//==============================================================
// 12) Servo enable and magnetic brake control
//==============================================================
// EN: Zero the movement request immediately, command quick stop and keep the
//     servo enabled only for the configured shutdown delay.
//     Drive-ready feedback is not used to avoid a circular enable dependency.
// PT: Zera a solicitação de movimento imediatamente, comanda o quick stop e
//     mantém o servo habilitado apenas durante o atraso configurado de desligamento.
//     O retorno de drive pronto não é usado para evitar dependência circular.
elevatorDriveEnableRequest :=
    systemRunEnable AND
    safetyCircuitOk;

tofElevatorDriveDisableDelay(
    IN := elevatorDriveEnableRequest,
    PT := machineConfig.elevatorDriveDisableDelay
);

elevatorDriveEnable :=
    tofElevatorDriveDisableDelay.Q;

elevatorQuickStop :=
    NOT elevatorDriveEnableRequest AND
    tofElevatorDriveDisableDelay.Q;

elevatorMoveRequest :=
    systemRunEnable AND
    safetyCircuitOk AND
    elevatorDriveOk AND
    NOT elevatorFault AND
    (ABS(elevatorSignedSpeedRefMmps) > 0.0);

IF elevatorMoveRequest THEN

    elevatorBrakeReleaseRequest := TRUE;
    tonElevatorBrakeHoldDelay(IN := FALSE);

ELSE

    IF elevatorBrakeRelease THEN

        tonElevatorBrakeHoldDelay(
            IN := TRUE,
            PT := machineConfig.elevatorBrakeHoldTime
        );

        elevatorBrakeReleaseRequest :=
            NOT tonElevatorBrakeHoldDelay.Q;

    ELSE

        tonElevatorBrakeHoldDelay(IN := FALSE);
        elevatorBrakeReleaseRequest := FALSE;

    END_IF

END_IF;

elevatorBrakeRelease :=
    systemRunEnable AND
    safetyCircuitOk AND
    elevatorDriveOk AND
    NOT elevatorFault AND
    elevatorBrakeReleaseRequest;

tonElevatorBrakeReleaseDelay(
    IN := elevatorMoveRequest AND elevatorBrakeRelease,
    PT := machineConfig.elevatorBrakeReleaseDelay
);


//==============================================================
// 12) Direction and speed outputs
//==============================================================
IF elevatorMoveRequest AND
   elevatorBrakeRelease AND
   tonElevatorBrakeReleaseDelay.Q THEN

    elevatorSpeedRefMmps := elevatorSignedSpeedRefMmps;
    elevatorRunUp := elevatorSignedSpeedRefMmps > 0.0;
    elevatorRunDown := elevatorSignedSpeedRefMmps < 0.0;

ELSE

    elevatorSpeedRefMmps := 0.0;
    elevatorRunUp := FALSE;
    elevatorRunDown := FALSE;

END_IF;
END_METHOD

METHOD _ExternalCommands : BOOL
VAR_INPUT
END_VAR
END_METHOD

//==============================================================
// COMPLEX STACKER — HMI STATUS
// EN: Maps internal status, outputs, positions and diagnostics
//     to the HMI status structure.
//==============================================================
METHOD _HmiStatus



//==============================================================
// 1) System general status
//==============================================================
hmiStatus.systemRunEnable :=
    systemRunEnable;

hmiStatus.safetyCircuitOk :=
    safetyCircuitOk;

hmiStatus.faultActive :=
    faultActive OR
    (
        backstopRequiredForAutomaticOperation AND
        backstopFault
    ) OR
    elevatorFault OR
    sheetStackDischargeFault OR
    sheetStackDischargeConveyorFault;

hmiStatus.deviceState :=
    deviceState;


//==============================================================
// 2) Sheet conveyor group status
//==============================================================
hmiStatus.synchronizedConveyorsRunning :=
    synchronizedConveyorsRunning;

hmiStatus.sheetConveyor1Run :=
    sheetConveyor1Run;

hmiStatus.sheetConveyor2Run :=
    sheetConveyor2Run;

hmiStatus.sheetConveyor3Run :=
    sheetConveyor3Run;

hmiStatus.sheetConveyor4Run :=
    sheetConveyor4Run;

hmiStatus.sheetConveyor1SpeedRefMPM :=
    sheetConveyor1SpeedRefMPM;

hmiStatus.sheetConveyor2SpeedRefMPM :=
    sheetConveyor2SpeedRefMPM;

hmiStatus.sheetConveyor3SpeedRefMPM :=
    sheetConveyor3SpeedRefMPM;

hmiStatus.sheetConveyor4SpeedRefMPM :=
    sheetConveyor4SpeedRefMPM;

hmiStatus.syncConveyorsState :=
    syncConveyorsState;


//==============================================================
// 3) Sheet stack separation status
//==============================================================
hmiStatus.sheetStackSeparationReady :=
    sheetStackSeparationReady;

hmiStatus.sheetStackSeparationActive :=
    sheetStackSeparationActive;

hmiStatus.sheetStackBrakeActive :=
    sheetStackBrakeActive;


//==============================================================
// 4) Sheet stack discharge sequence status
//==============================================================
hmiStatus.sheetStackDischargeState :=
    sheetStackDischargeState;

hmiStatus.sheetStackDischargeStateCode :=
    sheetStackDischargeStateCode;

hmiStatus.sheetStackDischargePending :=
    sheetStackDischargePending;

hmiStatus.sheetStackDischargeActive :=
    sheetStackDischargeActive;

hmiStatus.sheetStackDischargeStarted :=
    sheetStackDischargeStarted;

hmiStatus.sheetStackDischargeFinished :=
    sheetStackDischargeFinished;

hmiStatus.sheetStackDischargeFault :=
    sheetStackDischargeFault;

hmiStatus.sheetStackDischargeFaultCode :=
    sheetStackDischargeFaultCode;

hmiStatus.sheetStackDischargeLastCycleOk :=
    sheetStackDischargeLastCycleOk;

hmiStatus.sheetStackDischargeLastResultCode :=
    sheetStackDischargeLastResultCode;

hmiStatus.sheetStackDischargeLastFaultStepCode :=
    sheetStackDischargeLastFaultStepCode;

hmiStatus.sheetStackDischargeLastFaultCode :=
    sheetStackDischargeLastFaultCode;


//==============================================================
// 5) Sheet stack discharge conveyor status
//==============================================================
hmiStatus.sheetStackDischargeConveyorState :=
    sheetStackDischargeConveyorState;

hmiStatus.sheetStackDischargeConveyorRun :=
    sheetStackDischargeConveyorRun;

hmiStatus.sheetStackDischargeConveyorSpeedRefMPM :=
    sheetStackDischargeConveyorSpeedRefMPM;

hmiStatus.sheetStackDischargeConveyorFault :=
    sheetStackDischargeConveyorFault;

hmiStatus.sheetStackDischargeConveyorFaultCode :=
    sheetStackDischargeConveyorFaultCode;


//==============================================================
// 6) Backstop status
//==============================================================
hmiStatus.backstopState :=
    backstopState;

hmiStatus.backstopHomed :=
    backstopHomed;

hmiStatus.backstopHomeRunning :=
    backstopHomeRunning;

hmiStatus.backstopInPosition :=
    backstopInPosition;

hmiStatus.backstopPositionMm :=
    backstopPositionMm;

hmiStatus.backstopTargetPositionMm :=
    backstopTargetPositionMm;

hmiStatus.backstopPositionErrorMm :=
    backstopPositionErrorMm;

hmiStatus.backstopRunFw :=
    backstopRunFw;

hmiStatus.backstopRunRev :=
    backstopRunRev;

hmiStatus.backstopSpeedRefMmps :=
    backstopSpeedRefMmps;

hmiStatus.backstopPlateUpSolenoid :=
    backstopPlateUpSolenoid;

hmiStatus.backstopSetEncoderPosition :=
    backstopSetEncoderPosition;

hmiStatus.backstopSetEncoderPositionMm :=
    backstopSetEncoderPositionMm;

hmiStatus.backstopManualInterventionActive :=
    backstopManualInterventionActive;

hmiStatus.backstopManualInterventionPositionMm :=
    backstopManualInterventionPositionMm;

hmiStatus.backstopFault :=
    backstopFault;

hmiStatus.backstopFaultCode :=
    backstopFaultCode;


//==============================================================
// 7) Elevator status
//==============================================================
hmiStatus.elevatorState :=
    elevatorState;

hmiStatus.elevatorHomed :=
    elevatorHomed;

hmiStatus.elevatorInPosition :=
    elevatorInPosition;

hmiStatus.elevatorPositionMm :=
    elevatorPositionMm;

hmiStatus.elevatorTargetPositionMm :=
    elevatorTargetPositionMm;

hmiStatus.elevatorPositionErrorMm :=
    elevatorPositionErrorMm;

hmiStatus.elevatorRunUp :=
    elevatorRunUp;

hmiStatus.elevatorRunDown :=
    elevatorRunDown;

hmiStatus.elevatorBrakeRelease :=
    elevatorBrakeRelease;

hmiStatus.elevatorDriveEnable :=
    elevatorDriveEnable;

hmiStatus.elevatorQuickStop :=
    elevatorQuickStop;

hmiStatus.elevatorSpeedRefMmps :=
    elevatorSpeedRefMmps;

hmiStatus.elevatorSetEncoderPosition :=
    elevatorSetEncoderPosition;

hmiStatus.elevatorSetEncoderPositionMm :=
    elevatorSetEncoderPositionMm;

hmiStatus.elevatorFault :=
    elevatorFault;

hmiStatus.elevatorFaultCode :=
    elevatorFaultCode;


//==============================================================
// 8) Auxiliary pneumatic output status
// EN: Mirror the commanded pneumatic outputs for HMI diagnostics.
// PT: Espelha as saídas pneumáticas comandadas para diagnóstico na HMI.
//==============================================================
hmiStatus.paperPressSolenoid :=
    paperPressSolenoid;

hmiStatus.sheetBrush1Valve :=
    sheetBrush1Valve;

hmiStatus.sheetBrush2Valve :=
    sheetBrush2Valve;

hmiStatus.sheetBrush3Valve :=
    sheetBrush3Valve;

hmiStatus.sheetBrush4Valve :=
    sheetBrush4Valve;


//==============================================================
// 9) Process values
//==============================================================
hmiStatus.lineSpeedMPM :=
    lineSpeedMPM;

hmiStatus.sheetLengthMm :=
    sheetLengthMm;

hmiStatus.stackHeightMm :=
    stackHeightMm;


//==============================================================
// 10) Input / drive status mirror
//==============================================================
hmiStatus.sheetConveyor1DriveOk :=
    sheetConveyor1DriveOk;

hmiStatus.sheetConveyor2DriveOk :=
    sheetConveyor2DriveOk;

hmiStatus.sheetConveyor3DriveOk :=
    sheetConveyor3DriveOk;

hmiStatus.sheetConveyor4DriveOk :=
    sheetConveyor4DriveOk;

hmiStatus.backstopDriveOk :=
    backstopDriveOk;

hmiStatus.elevatorDriveOk :=
    elevatorDriveOk;

hmiStatus.sheetStackDischargeConveyorDriveOk :=
    sheetStackDischargeConveyorDriveOk;
END_METHOD

//==============================================================
// COMPLEX STACKER — MACHINE AUXILIARY CONTROL
// EN: Maps auxiliary outputs and generates external event pulses.
// PT: Mapeia saídas auxiliares e gera pulsos de eventos externos.
//==============================================================
METHOD _MachineAuxiliary

//==============================================================
// 1) Auxiliary pneumatic outputs
// EN: Maps the operator command to the no-crush roller valve.
// PT: Mapeia o comando do operador para a válvula dos rolos no-crush.
//==============================================================
noCrushRollersUpDownValve := noCrushRollersDownCmd;


//==============================================================
// 2) General status and command mirrors
// EN: Exposes the internal run and reset states to the parent controller.
// PT: Expõe os estados internos de operação e reset ao controlador pai.
//==============================================================
stackerRunning := systemRunEnable;
reset := resetCmd;


//==============================================================
// 3) Active unload and homing warning status
// EN: Includes pending separation so the warning starts in the acceptance
//     scan. Homing is detected from the current axis states so the siren
//     remains active throughout each complete homing sequence.
// PT: Inclui a separação pendente para o aviso iniciar no scan do aceite.
//     O homing é detectado pelos estados atuais dos eixos para manter a
//     sirene ativa durante toda a sequência de referenciamento.
//==============================================================
stackerBuzzer1 :=
    sheetStackDischargePending OR
    sheetStackDischargeActive OR
    (
        (backstopControlState >= 10) AND
        (backstopControlState <= 14)
    ) OR
    (
        (elevatorControlState >= 10) AND
        (elevatorControlState <= 14)
    );

stackerBuzzer2 :=
    sheetStackDischargePending OR
    sheetStackDischargeActive OR
    (
        (backstopControlState >= 10) AND
        (backstopControlState <= 14)
    ) OR
    (
        (elevatorControlState >= 10) AND
        (elevatorControlState <= 14)
    );

//==============================================================
// 4) External stack counter reset
// EN: Every accepted unload generates a fixed 20 ms reset pulse.
// PT: Cada descarga aceita gera um pulso fixo de reset de 20 ms.
//==============================================================
tpExternalCounterReset(
    IN := dischargeRequestAccepted,
    PT := T#20MS
);

externalCounterReset := tpExternalCounterReset.Q;
END_METHOD

METHOD _paperPressControl

// EN: When disabled, immediately switch off and reset the cycle.
// PT: Quando desabilitado, desliga imediatamente e reinicia o ciclo.
IF NOT paperPressAutoManCmd THEN

    paperPressSolenoid := FALSE;
    paperPressOnPhase := TRUE;


    instTONPaperPressOn(IN := FALSE);

    instTONPaperPressOff(IN := FALSE);


ELSE

	IF elevatorControlState = 30 THEN
		//==========================================================
		// ON phase / Fase ligada (Only when auto leveling)
		//==========================================================
		IF paperPressOnPhase THEN
	
			paperPressSolenoid := TRUE;
	
			instTONPaperPressOff(IN := FALSE);
	
			instTONPaperPressOn(
				IN := TRUE,
				PT := machineConfig.paperPressOnTime
			);
	
			IF instTONPaperPressOn.Q THEN
	
				instTONPaperPressOn(IN := FALSE);
	
				paperPressSolenoid := FALSE;
				paperPressOnPhase := FALSE;
	
			END_IF;
	
		//==========================================================
		// OFF phase / Fase desligada
		//==========================================================
		ELSE
	
			paperPressSolenoid := FALSE;
	
			instTONPaperPressOn(IN := FALSE);
	
			instTONPaperPressOff(
				IN := TRUE,
				PT := machineConfig.paperPressOffTime
			);
	
			IF instTONPaperPressOff.Q THEN
	
				instTONPaperPressOff(IN := FALSE);
	
				paperPressSolenoid := TRUE;
				paperPressOnPhase := TRUE;
	
			END_IF;
	
		END_IF;
		
	ELSE
		
		paperPressSolenoid := FALSE;
		paperPressOnPhase := TRUE;
	
	
		instTONPaperPressOn(IN := FALSE);
	
		instTONPaperPressOff(IN := FALSE);
	
	END_IF

END_IF;
END_METHOD

//==============================================================
// COMPLEX STACKER - SHEET BRUSH CONTROL
// EN: Controls the four independent sheet brushes from manual commands.
// PT: Controla as quatro escovas independentes pelos comandos manuais.
//==============================================================
METHOD _SheetBrushControl

// EN: The master command only enables the individual brush commands.
//     This function is intentionally independent of the stacker run state.
// PT: O comando mestre apenas habilita os comandos individuais das escovas.
//     Esta função é intencionalmente independente do estado ligado do stacker.
sheetBrush1Valve := sheetBrushAutoManCmd AND sheetBrush1Cmd;
sheetBrush2Valve := sheetBrushAutoManCmd AND sheetBrush2Cmd;
sheetBrush3Valve := sheetBrushAutoManCmd AND sheetBrush3Cmd;
sheetBrush4Valve := sheetBrushAutoManCmd AND sheetBrush4Cmd;
END_METHOD

//==============================================================
// COMPLEX STACKER - SHEET CONVEYOR 1 EXHAUST FAN CONTROL
// EN: Controls the exhaust fan according to stacker enable,
//     operator command and line speed.
// PT: Controla o exaustor conforme a habilitação do stacker,
//     o comando do operador e a velocidade da linha.
//==============================================================
METHOD _SheetConveyor1ExhaustFanControl

// EN: Operator disable or stacker shutdown switches the fan off immediately.
// PT: A desabilitação pelo operador ou o desligamento do stacker desliga
//     o exaustor imediatamente.
IF NOT systemRunEnable OR
   NOT sheetConveyor1ExhaustFanCmd THEN

    sheetConveyor1ExhaustFanRun := FALSE;
    instTONSheetConveyor1ExhaustFanStopDelay(IN := FALSE);

// EN: Above the configured threshold, run the fan and reset the stop delay.
// PT: Acima do limite configurado, liga o exaustor e reinicia o atraso.
ELSIF lineSpeedMPM > machineConfig.sheetConveyor1ExhaustFanLineSpeedThresholdMPM THEN

    sheetConveyor1ExhaustFanRun := TRUE;
    instTONSheetConveyor1ExhaustFanStopDelay(IN := FALSE);

// EN: When speed drops, keep an already running fan on until the delay expires.
//     Enabling the command at low speed does not start the fan.
// PT: Quando a velocidade cai, mantém o exaustor que já estava ligado até
//     o fim do atraso. Habilitar o comando em baixa velocidade não liga o exaustor.
ELSIF sheetConveyor1ExhaustFanRun THEN

    instTONSheetConveyor1ExhaustFanStopDelay(
        IN := TRUE,
        PT := machineConfig.sheetConveyor1ExhaustFanStopDelay
    );

    IF instTONSheetConveyor1ExhaustFanStopDelay.Q THEN

        sheetConveyor1ExhaustFanRun := FALSE;

    END_IF;

ELSE

    sheetConveyor1ExhaustFanRun := FALSE;
    instTONSheetConveyor1ExhaustFanStopDelay(IN := FALSE);

END_IF;
END_METHOD

//==============================================================
// COMPLEX STACKER — SHEET CONVEYOR GROUP CONTROL
// EN: Controls the synchronized sheet conveyor group.
//     Start/stop command latch is handled by _SystemControl().
//==============================================================
METHOD _SheetConveyorGroupControl

//==============================================================
// 1) Conditions
//==============================================================
// EN: Only synchronized sheet conveyor drives are considered here.
// PT: Apenas os inversores das esteiras sincronizadas são considerados aqui.
allSynchronizedDrivesOk :=
    sheetConveyor1DriveOk AND
    sheetConveyor2DriveOk AND
    sheetConveyor3DriveOk AND
    sheetConveyor4DriveOk;


// EN: Synchronized conveyor group fault.
// PT: Falha do grupo de esteiras sincronizadas.
anyFault :=
    NOT safetyCircuitOk OR
    NOT allSynchronizedDrivesOk;

faultActive := anyFault;


//==============================================================
// 2) State machine
//==============================================================
CASE syncConveyorsState OF

    0: // IDLE
        deviceState := 'IDLE';

        sheetConveyor1Run := FALSE;
        sheetConveyor2Run := FALSE;
        sheetConveyor3Run := FALSE;
        sheetConveyor4Run := FALSE;

        synchronizedConveyorsRunning := FALSE;

        // EN: The group starts only when the master system is enabled
        //     and no conveyor group fault is active.
        IF systemRunEnable AND NOT anyFault THEN

            syncConveyorsState := 1;

        ELSIF systemRunEnable AND anyFault THEN

            syncConveyorsState := 10;

        END_IF


    1: // RUN
        deviceState := 'RUN';

        // EN: Outputs are also directly conditioned by systemRunEnable
        //     to avoid one-scan movement after a stop command.
        sheetConveyor1Run :=
            systemRunEnable AND
            safetyCircuitOk AND
            sheetConveyor1DriveOk;

        sheetConveyor2Run :=
            systemRunEnable AND
            safetyCircuitOk AND
            sheetConveyor2DriveOk;

        sheetConveyor3Run :=
            systemRunEnable AND
            safetyCircuitOk AND
            sheetConveyor3DriveOk;

        sheetConveyor4Run :=
            systemRunEnable AND
            safetyCircuitOk AND
            sheetConveyor4DriveOk;

        synchronizedConveyorsRunning :=
            sheetConveyor1Run AND
            sheetConveyor2Run AND
            sheetConveyor3Run AND
            sheetConveyor4Run;

        IF anyFault THEN

            syncConveyorsState := 10;

        ELSIF NOT systemRunEnable THEN

            syncConveyorsState := 0;

        END_IF


    10: // FAULT
        deviceState := 'FAULT';

        sheetConveyor1Run := FALSE;
        sheetConveyor2Run := FALSE;
        sheetConveyor3Run := FALSE;
        sheetConveyor4Run := FALSE;

        synchronizedConveyorsRunning := FALSE;

        // EN: Fault state is released only by reset and with all faults cleared.
        //     If systemRunEnable is still TRUE after reset, the group can start
        //     again from IDLE on the next scan.
        IF resetCmd AND NOT anyFault THEN

            syncConveyorsState := 0;

        END_IF


ELSE

    syncConveyorsState := 0;

END_CASE;
END_METHOD

//==============================================================
// COMPLEX STACKER - SHEET STACK ALIGNMENT BRUSH CONTROL
// EN: Keeps the alignment brush engaged during production and raises
//     it only while the elevator executes an automatic discharge cycle.
// PT: Mantém a escova de alinhamento acionada durante a produção e a
//     levanta somente durante o ciclo automático de descarga do elevador.
//==============================================================
METHOD _SheetStackAlignmentBrushControl
VAR
	// EN: Relevant fault condition that forces the enabled brush down.
	// PT: Condição de falha relevante que força a escova habilitada para baixo.
	brushFaultActive : BOOL;
END_VAR


//==============================================================
// 2) Automatic discharge memory / Memória da descarga automática
//==============================================================
// EN: Manual operation and faults force the brush down and cancel the
//     memory of a previously active automatic discharge.
// PT: A operação manual e as falhas forçam a escova para baixo e cancelam
//     a memória de uma descarga automática anteriormente ativa.

    // EN: WAIT_SEPARATION (state 5) is intentionally excluded so the brush
    //     remains down until elevator discharge positioning actually starts.
    // PT: WAIT_SEPARATION (estado 5) é intencionalmente excluído para que a
    //     escova permaneça abaixada até iniciar o posicionamento de descarga.
    IF (sheetStackDischargeControlState = 10) OR
       (sheetStackDischargeControlState = 20) OR
       (sheetStackDischargeControlState = 30) OR
       (sheetStackDischargeControlState = 40) OR
       (sheetStackDischargeControlState = 50) THEN

        sheetStackAlignmentBrushLiftedForDischarge := TRUE;

    // EN: Lower the brush only after discharge has completely finished and
    //     automatic elevator leveling is active again.
    // PT: Abaixa a escova somente após o descarte terminar completamente e
    //     o nivelamento automático do elevador estar ativo novamente.
    ELSIF (sheetStackDischargeControlState = 0) AND
          NOT sheetStackDischargePending AND
          NOT sheetStackDischargeActive AND
          (elevatorControlState = 30) THEN

        sheetStackAlignmentBrushLiftedForDischarge := FALSE;

    END_IF


IF noCrushRollersDownCmd AND NOT sheetStackAlignmentBrushLiftedForDischarge THEN

	sheetStackAlignmentBrush := TRUE;

ELSE

	sheetStackAlignmentBrush := FALSE;

END_IF
END_METHOD

//==============================================================
// COMPLEX STACKER — SHEET STACK DISCHARGE CONTROL
// EN: Controls the sheet stack discharge sequence after the sheet
//     conveyor separation cycle is completed.
//
// State code
// 0  = IDLE
// 5  = WAIT_SEPARATION
// 10 = START_DISCHARGE_POSITIONING
// 20 = WAIT_DISCHARGE_POSITION
// 30 = RUN_DISCHARGE_CONVEYOR_AND_WAIT_CLEAR
// 40 = START_RETURN_POSITIONING
// 50 = WAIT_RETURN_POSITION
// 60 = FINISH
// 90 = FAULT_HOLD
//
// Last result code
// 0 = No cycle executed yet
// 1 = Last cycle completed successfully
// 2 = Last cycle completed with manual backstop skip
// 3 = Last cycle completed/aborted by timeout
// 4 = Last cycle aborted by fault
//
// Fault code
// 0  = No fault
// 1  = Safety circuit not OK
// 2  = Sheet conveyor drive not OK
// 3  = Discharge conveyor drive/control fault
// 4  = Backstop drive/control fault
// 5  = Elevator drive/control fault
// 6  = Stacker stopped during cycle
// 10 = Wait separation timeout
// 20 = Discharge positioning timeout
// 30 = Discharge conveyor did not start timeout
// 31 = Elevator platform clear timeout
// 50 = Return positioning timeout
//==============================================================
METHOD _SheetStackDischargeControl
VAR
    abortCycle : BOOL;
    automaticUnloadRequest : BOOL;
    changeBatchRequest : BOOL;
    backstopDischargeReady : BOOL;
    backstopAutomaticCycleEnabled : BOOL;
    elevatorPlatformClear : BOOL;
    restartFaultRecovery : BOOL;
    unloadRequestAvailable : BOOL;
END_VAR


//==============================================================
// 1) Default event pulses
//==============================================================
stackerUnloadAccepted       := FALSE;
dischargeRequestAccepted    := FALSE;
sheetStackDischargeStarted  := FALSE;
sheetStackDischargeFinished := FALSE;

// EN: An empty platform is accepted even when no stack was present
//     at the beginning of the discharge cycle.
// PT: Plataforma vazia é aceita mesmo quando não havia pilha
//     no início do ciclo de descarte.
elevatorPlatformClear :=
    NOT elevatorStackPresentAtDischargeStart OR
    (
        elevatorStackExitClearSensor AND
         elevatorStackPresentSensor
    );


//==============================================================
// 2) Default internal requests / overrides
//==============================================================
// EN: The sequence does not write the physical discharge conveyor outputs.
//     It only generates an internal request to the conveyor control method.
sheetStackDischargeConveyorRunRequest := FALSE;

backstopTargetOverrideActive := FALSE;
backstopTargetOverridePositionMm := 0.0;

elevatorTargetOverrideActive := FALSE;
elevatorTargetOverridePositionMm := 0.0;


//==============================================================
// 3) Unload request handling
//==============================================================
// EN: The local request is accepted only on its rising edge.
// PT: O pedido local é aceito somente na sua borda de subida.
rStackerUnloadCmd :=
    stackerUnloadCmd AND NOT stackerUnloadCmdOld;

stackerUnloadCmdOld := stackerUnloadCmd;


// EN: The maintained automatic request is rearmed only after going FALSE.
//     If it remains TRUE, it cannot be accepted for a second cycle.
// PT: O pedido automático mantido é rearmado somente após ficar FALSE.
//     Se permanecer TRUE, não pode ser aceito para um segundo ciclo.
IF NOT packageCompleteCmd THEN
    packageCompleteCmdAcceptedLatch := FALSE;
END_IF;

automaticUnloadRequest :=
    packageCompleteCmd AND
    NOT packageCompleteCmdAcceptedLatch;

// EN: Preserve a batch-change rising edge until the cycle can be accepted.
// PT: Preserva a borda de subida da troca de lote até o ciclo poder ser aceito.
IF changeBatchCmd AND
   NOT changeBatchCmdOld AND
   NOT automaticUnloadRequest THEN
    changeBatchRequestPending := TRUE;
END_IF;

changeBatchCmdOld := changeBatchCmd;
changeBatchRequest := changeBatchRequestPending;


// EN: The automatic request has priority when both requests arrive together.
// PT: O pedido automático tem prioridade quando os dois pedidos chegam juntos.
unloadRequestAvailable := FALSE;

IF automaticUnloadRequest THEN
    unloadRequestAvailable := TRUE;
    changeBatchRequest := FALSE;
ELSIF changeBatchRequest THEN
    unloadRequestAvailable := TRUE;
ELSIF rStackerUnloadCmd THEN
    unloadRequestAvailable := TRUE;
END_IF;


//==============================================================
// 3.1) Backstop participation in the current cycle
//==============================================================
// EN: Once manual mode is detected during an accepted cycle, keep the
//     backstop bypassed until that cycle finishes. Returning the selector
//     to automatic cannot restart an old backstop movement.
// PT: Depois que o modo manual for detectado durante um ciclo aceito,
//     mantém o backstop ignorado até o fim desse ciclo. Retornar o seletor
//     para automático não reinicia um movimento antigo do backstop.
IF (
       sheetStackDischargeActive OR
       sheetStackDischargePending OR
       (sheetStackDischargeControlState <> 0)
   ) AND
   NOT backstopAutoCmd THEN

    sheetStackDischargeCycleHasManualSkip := TRUE;

END_IF;


IF sheetStackDischargeActive OR
   sheetStackDischargePending OR
   (sheetStackDischargeControlState <> 0) THEN

    backstopAutomaticCycleEnabled :=
        backstopAutoCmd AND
        NOT sheetStackDischargeCycleHasManualSkip;

ELSE

    // EN: Before accepting a new cycle, use the current selector position.
    // PT: Antes de aceitar um novo ciclo, usa a posição atual do seletor.
    backstopAutomaticCycleEnabled := backstopAutoCmd;

END_IF;


//==============================================================
// 4) Fault condition
//==============================================================
// EN: Elevator drive, homing and position feedback are required
//     for safe discharge sequence progress.
// PT: Drive, homing e posição do elevador são obrigatórios
//     para o avanço seguro da sequência de descarte.
sheetStackDischargeFaultCondition :=
    NOT safetyCircuitOk OR
    NOT sheetConveyor1DriveOk OR
    NOT sheetConveyor2DriveOk OR
    NOT sheetConveyor3DriveOk OR
    NOT sheetConveyor4DriveOk OR
    NOT sheetStackDischargeConveyorDriveOk OR
    sheetStackDischargeConveyorFault OR
    (
        backstopAutomaticCycleEnabled AND
        (
            NOT backstopDriveOk OR
            NOT backstopHomed OR
            backstopFault
        )
    ) OR
    NOT elevatorDriveOk OR
    NOT elevatorHomed OR
    NOT elevatorReadyForAutomaticCycle OR
    elevatorFault;


//==============================================================
// 5) Fault code priority
//==============================================================
IF NOT safetyCircuitOk THEN

    sheetStackDischargeFaultCode := 1;

ELSIF NOT sheetConveyor1DriveOk OR
      NOT sheetConveyor2DriveOk OR
      NOT sheetConveyor3DriveOk OR
      NOT sheetConveyor4DriveOk THEN

    sheetStackDischargeFaultCode := 2;

ELSIF NOT sheetStackDischargeConveyorDriveOk OR
      sheetStackDischargeConveyorFault THEN

    sheetStackDischargeFaultCode := 3;

ELSIF backstopAutomaticCycleEnabled AND
      (
          NOT backstopDriveOk OR
          NOT backstopHomed OR
          backstopFault
      ) THEN

    sheetStackDischargeFaultCode := 4;

ELSIF NOT elevatorDriveOk OR
      NOT elevatorHomed OR
      NOT elevatorReadyForAutomaticCycle OR
      elevatorFault THEN

    sheetStackDischargeFaultCode := 5;

ELSIF NOT synchronizedConveyorsRunning THEN

    sheetStackDischargeFaultCode := 6;

END_IF;


//==============================================================
// 6) Optional reset of current sequence fault display
//==============================================================
// EN: Reset clears the current sequence fault flag,
//     but does not erase last cycle diagnostic codes.
IF resetCmd AND (sheetStackDischargeControlState = 0) THEN

    sheetStackDischargeFault := FALSE;
    sheetStackDischargeFaultCode := 0;
    changeBatchRequestPending := FALSE;
    changeBatchCycleActive := FALSE;

END_IF;


//==============================================================
// 7) Accept and arm the discharge sequence
//==============================================================
// EN: The request is accepted only when separation can start and every
//     discharge permissive is valid. A start-triggered homing request must
//     finish before a new discharge can be accepted.
// PT: O pedido é aceito somente quando a separação pode iniciar e todas as
//     permissões de descarga são válidas. Um homing solicitado pela partida
//     deve terminar antes que um novo descarte seja aceito.
IF unloadRequestAvailable AND
   sheetStackSeparationReady AND
   (packageSeparationState = 0) AND
   elevatorAutoCmd AND
   NOT elevatorAutoHomePending AND
   NOT (
       (elevatorControlState >= 10) AND
       (elevatorControlState <= 14)
   ) AND
   (
       NOT backstopAutoCmd OR
       (
           NOT backstopAutoHomePending AND
           NOT (
               (backstopControlState >= 10) AND
               (backstopControlState <= 14)
           )
       )
   ) AND
   synchronizedConveyorsRunning AND
   NOT sheetStackDischargeFaultCondition AND
   NOT sheetStackDischargeFault AND
   NOT sheetStackDischargeActive AND
   NOT sheetStackDischargePending THEN

    sheetStackDischargePending := TRUE;
    dischargeRequestAccepted := TRUE;

    // EN: Consume the automatic request until packageCompleteCmd turns FALSE.
    //     This branch also implements automatic priority over the local edge.
    // PT: Consome o pedido automático até packageCompleteCmd ficar FALSE.
    //     Este ramo também implementa a prioridade do automático sobre a borda local.
    IF automaticUnloadRequest THEN
        packageCompleteCmdAcceptedLatch := TRUE;
        changeBatchCycleActive := FALSE;
    ELSIF changeBatchRequest THEN
        changeBatchRequestPending := FALSE;
        changeBatchCycleActive := TRUE;
    ELSE
        changeBatchCycleActive := FALSE;
        stackerUnloadAccepted := TRUE;
    END_IF;

    // EN: Clear current-cycle flags when a new cycle is accepted.
    sheetStackDischargeFault := FALSE;
    sheetStackDischargeFaultCode := 0;

    // EN: Manual is a valid bypass. It remains latched for this whole cycle.
    // PT: Manual é um bypass válido. Permanece memorizado por todo o ciclo.
    sheetStackDischargeCycleHasManualSkip := NOT backstopAutoCmd;
    sheetStackDischargeCycleHasTimeout := FALSE;

END_IF;


//==============================================================
// 8) Start-triggered recovery from fault hold
//==============================================================
// EN: A new machine start safely abandons the failed discharge cycle before
//     the mandatory automatic homing requests are released on the next scan.
//     Last-cycle diagnostic codes and the accepted package latch are preserved.
// PT: Uma nova partida da máquina abandona com segurança o ciclo de descarte
//     com falha antes de liberar os pedidos obrigatórios de homing no próximo scan.
//     Os diagnósticos do último ciclo e o latch do pacote aceito são preservados.
restartFaultRecovery :=
    rStartCmd AND
    systemRunEnable AND
    (sheetStackDischargeControlState = 90);


IF restartFaultRecovery THEN

    sheetStackDischargeActive := FALSE;
    sheetStackDischargePending := FALSE;
    sheetStackDischargeControlState := 0;

    sheetStackDischargeFault := FALSE;
    sheetStackDischargeFaultCode := 0;
    changeBatchCycleActive := FALSE;

    sheetStackDischargeConveyorRunRequest := FALSE;

    backstopTargetOverrideActive := FALSE;
    elevatorTargetOverrideActive := FALSE;

    tonSheetStackDischarge(IN := FALSE);
    tonSheetStackDischargeStepTimeout(IN := FALSE);
    tonSheetStackDischargePlatformClearTimeout(IN := FALSE);

    elevatorPlatformClearDetected := FALSE;
    elevatorStackPresentAtDischargeStart := FALSE;

END_IF;


//==============================================================
// 9) Immediate abort condition
//==============================================================
// EN: Faults before discharge positioning cancel the request. Faults after
//     positioning starts hold safe targets until operator acknowledgement.
// PT: Falhas antes do posicionamento cancelam o pedido. Após o início,
//     mantêm os alvos seguros até o reconhecimento do operador.
abortCycle :=
    (
        sheetStackDischargeActive OR
        sheetStackDischargePending OR
        (sheetStackDischargeControlState <> 0)
    )
    AND
    (
        sheetStackDischargeFaultCondition OR
        NOT synchronizedConveyorsRunning
    );


IF abortCycle THEN

    sheetStackDischargeConveyorRunRequest := FALSE;
    sheetStackDischargePending := FALSE;
    changeBatchCycleActive := FALSE;

    tonSheetStackDischarge(IN := FALSE);
    tonSheetStackDischargeStepTimeout(IN := FALSE);
    tonSheetStackDischargePlatformClearTimeout(IN := FALSE);

    sheetStackDischargeFault := TRUE;

    sheetStackDischargeLastCycleOk := FALSE;
    sheetStackDischargeLastResultCode := 4;
    sheetStackDischargeLastFaultCode := sheetStackDischargeFaultCode;

    // EN: Do not clear backstopManualInterventionActive here.
    //     If the cycle aborted before return, keeping the memory is safer
    //     for the next cycle.

    IF sheetStackDischargeControlState <= 5 THEN

        // EN: No discharge movement has started yet.
        // PT: Nenhum movimento de descarte foi iniciado.
        sheetStackDischargeActive := FALSE;

        backstopTargetOverrideActive := FALSE;
        elevatorTargetOverrideActive := FALSE;

        elevatorPlatformClearDetected := FALSE;
        elevatorStackPresentAtDischargeStart := FALSE;

        sheetStackDischargeLastFaultStepCode :=
            sheetStackDischargeControlState;

        sheetStackDischargeState := 'ABORTED';
        sheetStackDischargeStateCode := 90;
        sheetStackDischargeControlState := 0;

    ELSE

        // EN: Preserve the original failed step while the external
        //     fault condition remains active in FAULT_HOLD.
        // PT: Preserva o passo original da falha enquanto a condição
        //     externa permanecer ativa no FAULT_HOLD.
        IF sheetStackDischargeControlState <> 90 THEN
            sheetStackDischargeLastFaultStepCode :=
                sheetStackDischargeControlState;
        END_IF;

        sheetStackDischargeActive := TRUE;
        sheetStackDischargeState := 'FAULT_HOLD';
        sheetStackDischargeStateCode := 90;

        IF sheetStackDischargeLastFaultStepCode < 40 THEN

            IF backstopAutomaticCycleEnabled THEN

                backstopTargetOverrideActive := TRUE;
                backstopTargetOverridePositionMm :=
                    backstopDischargeOpenTargetMm;

            END_IF;

            elevatorTargetOverrideActive := TRUE;
            elevatorTargetOverridePositionMm :=
                machineConfig.elevatorMinPositionMm;

        ELSE

            IF backstopAutomaticCycleEnabled THEN

                backstopTargetOverrideActive := TRUE;
                backstopTargetOverridePositionMm :=
                    backstopProgrammedDischargeTargetMm;

            END_IF;

            elevatorTargetOverrideActive := TRUE;
            elevatorTargetOverridePositionMm :=
                machineConfig.elevatorMaxPositionMm;

        END_IF;

        sheetStackDischargeControlState := 90;

    END_IF


ELSE

    //==============================================================
    // 10) Sheet stack discharge state machine
    //==============================================================
    CASE sheetStackDischargeControlState OF

        0: // IDLE
            sheetStackDischargeState := 'IDLE';
            sheetStackDischargeStateCode := 0;

            sheetStackDischargeActive := FALSE;

            sheetStackDischargeConveyorRunRequest := FALSE;

            backstopTargetOverrideActive := FALSE;
            elevatorTargetOverrideActive := FALSE;

            tonSheetStackDischarge(IN := FALSE);
            tonSheetStackDischargeStepTimeout(IN := FALSE);
            tonSheetStackDischargePlatformClearTimeout(IN := FALSE);
            elevatorPlatformClearDetected := FALSE;
            elevatorStackPresentAtDischargeStart := FALSE;

            IF sheetStackDischargePending THEN

                tonSheetStackDischarge(IN := FALSE);
                tonSheetStackDischargeStepTimeout(IN := FALSE);

                sheetStackDischargeControlState := 5;

            END_IF


        5: // WAIT_SEPARATION
            sheetStackDischargeState := 'WAIT_SEPARATION';
            sheetStackDischargeStateCode := 5;

            sheetStackDischargeActive := FALSE;

            sheetStackDischargeConveyorRunRequest := FALSE;

            backstopTargetOverrideActive := FALSE;
            elevatorTargetOverrideActive := FALSE;

            tonSheetStackDischarge(IN := FALSE);

            // EN: Wait for conveyor speed control to finish sheet stack separation.
            tonSheetStackDischargeStepTimeout(
                IN := TRUE,
                PT := machineConfig.sheetStackDischargeWaitSeparationTimeout
            );

            // EN: Complex stacker discharge starts only after conveyor 4
            //     completes the package separation sequence.
            // PT: O descarte do stacker complexo inicia somente depois que
            //     a esteira 4 concluir a sequência de separação do pacote.
            IF sheetStackSeparationFinished AND
               sheetConveyor4SeparationFinished THEN

                tonSheetStackDischargeStepTimeout(IN := FALSE);

                sheetStackDischargeControlState := 10;


            ELSIF tonSheetStackDischargeStepTimeout.Q THEN

                // EN: Separation did not finish. Do not discharge.
                tonSheetStackDischargeStepTimeout(IN := FALSE);

                sheetStackDischargePending := FALSE;
                sheetStackDischargeActive := FALSE;
                changeBatchCycleActive := FALSE;

                sheetStackDischargeFault := TRUE;
                sheetStackDischargeFaultCode := 10;

                sheetStackDischargeLastCycleOk := FALSE;
                sheetStackDischargeLastResultCode := 3;
                sheetStackDischargeLastFaultStepCode := 5;
                sheetStackDischargeLastFaultCode := 10;

                sheetStackDischargeControlState := 0;

            END_IF


        10: // START_DISCHARGE_POSITIONING
            sheetStackDischargeState := 'START_POSITIONING';
            sheetStackDischargeStateCode := 10;

            sheetStackDischargePending := FALSE;
            sheetStackDischargeActive := TRUE;
            sheetStackDischargeStarted := TRUE;

            elevatorPlatformClearDetected := FALSE;
            tonSheetStackDischargePlatformClearTimeout(IN := FALSE);
            elevatorStackPresentAtDischargeStart :=
                elevatorStackPresentSensor;

            tonSheetStackDischarge(IN := FALSE);
            tonSheetStackDischargeStepTimeout(IN := FALSE);

            //======================================================
            // EN: Latch programmed backstop target for this cycle.
            //     This is the normal position based on sheet length.
            //======================================================
            backstopProgrammedDischargeTargetMm :=
                LIMIT(
                    machineConfig.backstopMinPositionMm,
                    MAX(0.0, sheetLengthMm) +
                        machineConfig.backstopSheetLengthOffsetMm,
                    machineConfig.backstopMaxPositionMm
                );

            //======================================================
            // EN: Define safe opening base position.
            //     The opening starts from the actual mechanical position,
            //     independently of a new, smaller programmed sheet length.
            // PT: Define a posição base segura para abertura.
            //     A abertura parte da posição mecânica atual, independente
            //     de uma nova medida programada menor para a chapa.
            //======================================================
            backstopDischargeOpenBasePositionMm :=
                backstopPositionMm;

            IF backstopManualInterventionActive THEN

                backstopDischargeOpenBasePositionMm :=
                    MAX(
                        backstopDischargeOpenBasePositionMm,
                        backstopManualInterventionPositionMm
                    );

            END_IF;

            //======================================================
            // EN: Latch safe discharge open target.
            //     Only a non-negative offset is accepted.
            // PT: Memoriza o alvo seguro de abertura para descarga.
            //     Somente um offset não negativo é aceito.
            //======================================================
            backstopDischargeOpenTargetMm :=
                LIMIT(
                    machineConfig.backstopMinPositionMm,
                    backstopDischargeOpenBasePositionMm +
                        MAX(
                            0.0,
                            machineConfig.backstopDischargeOpenOffsetMm
                        ),
                    machineConfig.backstopMaxPositionMm
                );

            // EN: Request safe backstop opening only when it participates
            //     in the current automatic cycle. Manual mode is bypassed.
            // PT: Solicita a abertura segura do backstop somente quando ele
            //     participa do ciclo automático atual. O modo manual é ignorado.
            IF backstopAutomaticCycleEnabled THEN

                backstopTargetOverrideActive := TRUE;
                backstopTargetOverridePositionMm :=
                    backstopDischargeOpenTargetMm;

            END_IF;

            // EN: Request the elevator lower discharge position.
            // PT: Solicita a posição inferior de descarte do elevador.
            elevatorTargetOverrideActive := TRUE;
            elevatorTargetOverridePositionMm :=
                machineConfig.elevatorMinPositionMm;

            sheetStackDischargeControlState := 20;


        20: // WAIT_DISCHARGE_POSITION
            sheetStackDischargeState := 'WAIT_DISCHARGE_POS';
            sheetStackDischargeStateCode := 20;

            sheetStackDischargeActive := TRUE;

            // EN: In manual mode do not command or wait for the backstop.
            // PT: No modo manual não comanda nem aguarda o backstop.
            IF backstopAutomaticCycleEnabled THEN

                backstopTargetOverrideActive := TRUE;
                backstopTargetOverridePositionMm :=
                    backstopDischargeOpenTargetMm;

                backstopDischargeReady := backstopInPosition;

            ELSE

                backstopTargetOverrideActive := FALSE;
                backstopDischargeReady := TRUE;

            END_IF;

            // EN: Keep the lower discharge target active and wait for feedback.
            // PT: Mantém o alvo inferior de descarte e aguarda o feedback.
            elevatorTargetOverrideActive := TRUE;
            elevatorTargetOverridePositionMm :=
                machineConfig.elevatorMinPositionMm;

            IF backstopDischargeReady AND elevatorInPosition THEN

                tonSheetStackDischargeStepTimeout(IN := FALSE);
                sheetStackDischargeControlState := 30;

            ELSE

                tonSheetStackDischargeStepTimeout(
                    IN := TRUE,
                    PT := machineConfig.sheetStackDischargePositioningTimeout
                );

                IF tonSheetStackDischargeStepTimeout.Q THEN

                    tonSheetStackDischargeStepTimeout(IN := FALSE);

                    sheetStackDischargeCycleHasTimeout := TRUE;
                    sheetStackDischargeFault := TRUE;
                    sheetStackDischargeFaultCode := 20;

                    sheetStackDischargeLastCycleOk := FALSE;
                    sheetStackDischargeLastResultCode := 3;
                    sheetStackDischargeLastFaultStepCode := 20;
                    sheetStackDischargeLastFaultCode := 20;

                    // EN: Do not start the discharge conveyor without
                    //     confirmed elevator positioning.
                    // PT: Não inicia a esteira de descarte sem confirmar
                    //     o posicionamento do elevador.
                    sheetStackDischargeControlState := 90;
                    sheetStackDischargeActive := TRUE;
                    sheetStackDischargePending := FALSE;

                END_IF

            END_IF


        30: // RUN_DISCHARGE_CONVEYOR
            sheetStackDischargeState := 'DISCHARGING';
            sheetStackDischargeStateCode := 30;

            sheetStackDischargeActive := TRUE;

            // EN: Keep the backstop open only if it participates in this cycle.
            // PT: Mantém o backstop aberto somente se ele participa deste ciclo.
            IF backstopAutomaticCycleEnabled THEN

                backstopTargetOverrideActive := TRUE;
                backstopTargetOverridePositionMm :=
                    backstopDischargeOpenTargetMm;

            END_IF;

            // EN: Keep elevator at the lower discharge position.
            // PT: Mantém o elevador na posição inferior de descarte.
            elevatorTargetOverrideActive := TRUE;
            elevatorTargetOverridePositionMm :=
                machineConfig.elevatorMinPositionMm;

            // EN: Request discharge conveyor run.
            //     Physical output is controlled by _SheetStackDischargeConveyorControl.
            sheetStackDischargeConveyorRunRequest := TRUE;

            // EN: If conveyor is not actually running, use start timeout.
            IF NOT sheetStackDischargeConveyorRun THEN

                tonSheetStackDischarge(IN := FALSE);
                tonSheetStackDischargePlatformClearTimeout(IN := FALSE);

                tonSheetStackDischargeStepTimeout(
                    IN := TRUE,
                    PT := machineConfig.sheetStackDischargeConveyorStartTimeout
                );

                IF tonSheetStackDischargeStepTimeout.Q THEN

                    // EN: Conveyor did not start. Do not stay trapped.
                    tonSheetStackDischargeStepTimeout(IN := FALSE);

                    sheetStackDischargeConveyorRunRequest := FALSE;

                    sheetStackDischargeCycleHasTimeout := TRUE;

                    sheetStackDischargeFault := TRUE;
                    sheetStackDischargeFaultCode := 30;

                    sheetStackDischargeLastCycleOk := FALSE;
                    sheetStackDischargeLastResultCode := 3;
                    sheetStackDischargeLastFaultStepCode := 30;
                    sheetStackDischargeLastFaultCode := 30;

                    sheetStackDischargeControlState := 90;

                END_IF


            ELSE

                // EN: Conveyor is running. Count minimum discharge time
                //     and wait for a clean elevator platform.
                // PT: A esteira está em movimento. Conta o tempo mínimo
                //     e aguarda a plataforma do elevador ficar livre.
                tonSheetStackDischargeStepTimeout(IN := FALSE);

                tonSheetStackDischarge(
                    IN := TRUE,
                    PT := machineConfig.sheetStackDischargeTime
                );

                IF elevatorPlatformClear THEN
                    elevatorPlatformClearDetected := TRUE;
                END_IF;

                tonSheetStackDischargePlatformClearTimeout(
                    IN := NOT elevatorPlatformClearDetected,
                    PT := machineConfig.sheetStackDischargePlatformClearTimeout
                );

                IF tonSheetStackDischarge.Q AND
                   elevatorPlatformClearDetected THEN

                    tonSheetStackDischarge(IN := FALSE);
                    tonSheetStackDischargePlatformClearTimeout(IN := FALSE);

                    sheetStackDischargeConveyorRunRequest := FALSE;

                    sheetStackDischargeControlState := 40;

                ELSIF tonSheetStackDischargePlatformClearTimeout.Q THEN

                    tonSheetStackDischarge(IN := FALSE);
                    tonSheetStackDischargePlatformClearTimeout(IN := FALSE);

                    sheetStackDischargeConveyorRunRequest := FALSE;

                    sheetStackDischargeCycleHasTimeout := TRUE;
                    sheetStackDischargeFault := TRUE;
                    sheetStackDischargeFaultCode := 31;

                    sheetStackDischargeLastCycleOk := FALSE;
                    sheetStackDischargeLastResultCode := 3;
                    sheetStackDischargeLastFaultStepCode := 30;
                    sheetStackDischargeLastFaultCode := 31;

                    // EN: Keep the elevator down and backstop open until reset.
                    // PT: Mantém o elevador embaixo e o backstop aberto até o reset.
                    sheetStackDischargeControlState := 90;

                END_IF

            END_IF


        40: // START_RETURN_POSITIONING
            sheetStackDischargeState := 'START_RETURN';
            sheetStackDischargeStateCode := 40;

            sheetStackDischargeActive := TRUE;

            sheetStackDischargeConveyorRunRequest := FALSE;

            tonSheetStackDischarge(IN := FALSE);
            tonSheetStackDischargeStepTimeout(IN := FALSE);

            // EN: Return the backstop only if it participates in this cycle.
            // PT: Retorna o backstop somente se ele participa deste ciclo.
            IF backstopAutomaticCycleEnabled THEN

                backstopTargetOverrideActive := TRUE;
                backstopTargetOverridePositionMm :=
                    backstopProgrammedDischargeTargetMm;

            END_IF;

            // EN: Request elevator return to the upper production position.
            // PT: Solicita o retorno do elevador à posição superior de produção.
            elevatorTargetOverrideActive := TRUE;
            elevatorTargetOverridePositionMm :=
                machineConfig.elevatorMaxPositionMm;

            sheetStackDischargeControlState := 50;


        50: // WAIT_RETURN_POSITION
            sheetStackDischargeState := 'WAIT_RETURN_POS';
            sheetStackDischargeStateCode := 50;

            sheetStackDischargeActive := TRUE;

            sheetStackDischargeConveyorRunRequest := FALSE;

            // EN: In manual mode do not command or wait for backstop return.
            // PT: No modo manual não comanda nem aguarda o retorno do backstop.
            IF backstopAutomaticCycleEnabled THEN

                backstopTargetOverrideActive := TRUE;
                backstopTargetOverridePositionMm :=
                    backstopProgrammedDischargeTargetMm;

                backstopDischargeReady := backstopInPosition;

            ELSE

                backstopTargetOverrideActive := FALSE;
                backstopDischargeReady := TRUE;

            END_IF;

            // EN: Keep the upper elevator target active and wait for feedback.
            // PT: Mantém o alvo superior do elevador e aguarda o feedback.
            elevatorTargetOverrideActive := TRUE;
            elevatorTargetOverridePositionMm :=
                machineConfig.elevatorMaxPositionMm;

            IF backstopDischargeReady AND elevatorInPosition THEN

                tonSheetStackDischargeStepTimeout(IN := FALSE);
                sheetStackDischargeControlState := 60;

            ELSE

                tonSheetStackDischargeStepTimeout(
                    IN := TRUE,
                    PT := machineConfig.sheetStackDischargeReturnTimeout
                );

                IF tonSheetStackDischargeStepTimeout.Q THEN

                    tonSheetStackDischargeStepTimeout(IN := FALSE);

                    sheetStackDischargeCycleHasTimeout := TRUE;
                    sheetStackDischargeFault := TRUE;
                    sheetStackDischargeFaultCode := 50;

                    sheetStackDischargeLastCycleOk := FALSE;
                    sheetStackDischargeLastResultCode := 3;
                    sheetStackDischargeLastFaultStepCode := 50;
                    sheetStackDischargeLastFaultCode := 50;

                    // EN: Do not report a completed cycle without confirmed
                    //     return positioning.
                    // PT: Não confirma o ciclo sem o posicionamento de retorno.
                    sheetStackDischargeActive := TRUE;
                    sheetStackDischargePending := FALSE;
                    sheetStackDischargeControlState := 90;

                END_IF

            END_IF


        90: // FAULT_HOLD
            sheetStackDischargeState := 'FAULT_HOLD';
            sheetStackDischargeStateCode := 90;

            sheetStackDischargeActive := TRUE;
            sheetStackDischargePending := FALSE;
            sheetStackDischargeConveyorRunRequest := FALSE;

            tonSheetStackDischarge(IN := FALSE);
            tonSheetStackDischargeStepTimeout(IN := FALSE);
            tonSheetStackDischargePlatformClearTimeout(IN := FALSE);

            // EN: Before platform clearance, keep the safe discharge
            //     positions: backstop open and elevator down.
            // PT: Antes da confirmação de plataforma livre, mantém as
            //     posições seguras: backstop aberto e elevador embaixo.
            IF sheetStackDischargeLastFaultStepCode < 40 THEN

                IF backstopAutomaticCycleEnabled THEN

                    backstopTargetOverrideActive := TRUE;
                    backstopTargetOverridePositionMm :=
                        backstopDischargeOpenTargetMm;

                END_IF;

                elevatorTargetOverrideActive := TRUE;
                elevatorTargetOverridePositionMm :=
                    machineConfig.elevatorMinPositionMm;

            ELSE

                // EN: A return-position timeout occurs only after the
                //     platform was confirmed clear. Keep the return targets.
                // PT: Timeout de retorno ocorre somente após confirmar a
                //     plataforma livre. Mantém os alvos de retorno.
                IF backstopAutomaticCycleEnabled THEN

                    backstopTargetOverrideActive := TRUE;
                    backstopTargetOverridePositionMm :=
                        backstopProgrammedDischargeTargetMm;

                END_IF;

                elevatorTargetOverrideActive := TRUE;
                elevatorTargetOverridePositionMm :=
                    machineConfig.elevatorMaxPositionMm;

            END_IF;

            // EN: Reset is an explicit operator acknowledgement.
            // PT: Reset é uma confirmação explícita do operador.
            IF resetCmd AND
               safetyCircuitOk AND
               (
                   NOT backstopAutomaticCycleEnabled OR
                   backstopDriveOk
               ) AND
               elevatorDriveOk AND
               (
                   elevatorPlatformClear OR
                   elevatorPlatformClearDetected OR
                   (sheetStackDischargeLastFaultStepCode >= 40)
               ) THEN

                sheetStackDischargeFault := FALSE;
                sheetStackDischargeFaultCode := 0;

                // EN: After acknowledgement, complete the automatic return
                //     instead of releasing production immediately.
                // PT: Após o reconhecimento, conclui o retorno automático
                //     antes de liberar novamente a produção.
                sheetStackDischargeControlState := 40;

            END_IF


        60: // FINISH
            sheetStackDischargeState := 'FINISH';
            sheetStackDischargeStateCode := 60;

            sheetStackDischargeActive := FALSE;
            sheetStackDischargePending := FALSE;
            sheetStackDischargeFinished := TRUE;
            changeBatchCycleActive := FALSE;

            sheetStackDischargeConveyorRunRequest := FALSE;

            backstopTargetOverrideActive := FALSE;
            elevatorTargetOverrideActive := FALSE;

            tonSheetStackDischarge(IN := FALSE);
            tonSheetStackDischargeStepTimeout(IN := FALSE);
            tonSheetStackDischargePlatformClearTimeout(IN := FALSE);
            elevatorPlatformClearDetected := FALSE;
            elevatorStackPresentAtDischargeStart := FALSE;

            IF sheetStackDischargeCycleHasTimeout THEN

                sheetStackDischargeLastCycleOk := FALSE;
                sheetStackDischargeLastResultCode := 3;

                // EN: Keep manual intervention memory after timeout.
                //     The backstop may not have returned correctly.

            ELSIF sheetStackDischargeCycleHasManualSkip THEN

                sheetStackDischargeLastCycleOk := FALSE;
                sheetStackDischargeLastResultCode := 2;
                sheetStackDischargeLastFaultStepCode := 0;
                sheetStackDischargeLastFaultCode := 0;

                sheetStackDischargeFault := FALSE;
                sheetStackDischargeFaultCode := 0;

                // EN: Keep manual intervention memory because the backstop
                //     was not controlled automatically.


            ELSE

                sheetStackDischargeLastCycleOk := TRUE;
                sheetStackDischargeLastResultCode := 1;
                sheetStackDischargeLastFaultStepCode := 0;
                sheetStackDischargeLastFaultCode := 0;

                sheetStackDischargeFault := FALSE;
                sheetStackDischargeFaultCode := 0;

                // EN: Cycle completed correctly and backstop returned to
                //     programmed target. Clear manual intervention memory.
                backstopManualInterventionActive := FALSE;
                backstopManualInterventionPositionMm := 0.0;

            END_IF

            // EN: Always return to IDLE automatically.
            sheetStackDischargeControlState := 0;


    ELSE

        changeBatchCycleActive := FALSE;
        sheetStackDischargeControlState := 0;

    END_CASE;

END_IF;
END_METHOD

//==============================================================
// COMPLEX STACKER — SHEET STACK DISCHARGE CONVEYOR CONTROL
// EN: Controls the sheet stack discharge conveyor.
//     Conveyor runs while manual button is pressed or while
//     automatic request is active and conveyor automatic mode is enabled.
//
// Fault code
// 0 = No fault
// 1 = Safety circuit not OK
// 2 = Discharge conveyor drive not OK
//==============================================================
METHOD _SheetStackDischargeConveyorControl
VAR
    manualRunRequest   : BOOL;
    automaticRunRequest: BOOL;
    finalRunRequest    : BOOL;
END_VAR
//==============================================================
// COMPLEX STACKER — SHEET STACK DISCHARGE CONVEYOR CONTROL
// EN: Controls the sheet stack discharge conveyor in manual pulse
//     or automatic sequence request.
//==============================================================


//==============================================================
// 1) Default outputs
//==============================================================
sheetStackDischargeConveyorRun := FALSE;
sheetStackDischargeConveyorSpeedRefMPM := 0.0;


//==============================================================
// 2) Run request selection
//==============================================================
// EN: Manual command is momentary. The conveyor runs while its dedicated
//     button is pressed or while a valid, rearmed elevator down command remains
//     pressed after the elevator reaches the configured minimum position.
// PT: O comando manual é momentâneo. A esteira gira enquanto seu botão
//     dedicado estiver pressionado ou enquanto um comando de descida válido e
//     rearmado permanecer pressionado após atingir a posição mínima configurada.
manualRunRequest :=
    sheetStackDischargeConveyorManualRunCmd OR
    (
        elevatorManualCommandRequest AND
        elevatorDownCmd AND
        NOT elevatorUpCmd AND
        elevatorAtMinPosition AND
        (sheetStackDischargeControlState = 0) AND
        NOT elevatorFault AND
        NOT elevatorLowerSafetyLimit
    );


// EN: Automatic request is generated by the discharge sequence or by the
//     elevator homing platform-clear step.
// PT: O pedido automático é gerado pela sequência de descarga ou pela etapa
//     de limpeza da plataforma durante o homing do elevador.
automaticRunRequest :=
    sheetStackDischargeConveyorRunRequest OR
    elevatorHomeDischargeConveyorRunRequest;


// EN: Master system enable blocks both manual and automatic movement.
finalRunRequest :=
    systemRunEnable AND
    (
        manualRunRequest OR
        automaticRunRequest
    );


//==============================================================
// 3) Fault detection
//==============================================================
IF NOT safetyCircuitOk THEN

    sheetStackDischargeConveyorState := 'SAFETY_OFF';

    sheetStackDischargeConveyorFault := TRUE;
    sheetStackDischargeConveyorFaultCode := 1;


ELSIF NOT sheetStackDischargeConveyorDriveOk THEN

    sheetStackDischargeConveyorState := 'DRIVE_NOT_OK';

    sheetStackDischargeConveyorFault := TRUE;
    sheetStackDischargeConveyorFaultCode := 2;


ELSE

    //==============================================================
    // 4) Fault reset
    //==============================================================
    IF resetCmd THEN

        sheetStackDischargeConveyorFault := FALSE;
        sheetStackDischargeConveyorFaultCode := 0;

    END_IF;


    //==============================================================
    // 5) Conveyor output control
    //==============================================================
    IF sheetStackDischargeConveyorFault THEN

        sheetStackDischargeConveyorState := 'FAULT';

        sheetStackDischargeConveyorRun := FALSE;
        sheetStackDischargeConveyorSpeedRefMPM := 0.0;


    ELSIF NOT systemRunEnable THEN

        // EN: Master stop disables movement without generating a conveyor fault.
        sheetStackDischargeConveyorState := 'SYSTEM_DISABLED';

        sheetStackDischargeConveyorRun := FALSE;
        sheetStackDischargeConveyorSpeedRefMPM := 0.0;


    ELSIF finalRunRequest THEN

        IF automaticRunRequest THEN

            sheetStackDischargeConveyorState := 'AUTO_RUN';

        ELSE

            sheetStackDischargeConveyorState := 'MANUAL_RUN';

        END_IF;

        sheetStackDischargeConveyorRun := TRUE;

        sheetStackDischargeConveyorSpeedRefMPM :=
            LIMIT(
                0.0,
                machineConfig.sheetStackDischargeConveyorSpeedMPM,
                machineConfig.maximumSpeedMPM
            );


    ELSE

        sheetStackDischargeConveyorState := 'STOP';

        sheetStackDischargeConveyorRun := FALSE;
        sheetStackDischargeConveyorSpeedRefMPM := 0.0;

    END_IF

END_IF;
END_METHOD

//==============================================================
// COMPLEX STACKER - STACK BUFFER CONVEYOR CONTROL
// EN: Transfers finished stacks to the furthest available buffer.
// PT: Transfere as pilhas prontas para o buffer livre mais distante.
//==============================================================
METHOD _StackBufferConveyorsControl
VAR
    allBufferDrivesOk : BOOL;
    automaticTransferActive : BOOL;
END_VAR
//==============================================================
// 1) Common conditions and edge detection
//==============================================================
// EN: Default one-scan timeout event.
// PT: Evento padrão de timeout com duração de um scan.
stackBufferTransferTimeoutPulse := FALSE;


allBufferDrivesOk :=
    stackBufferConveyor1DriveOk AND
    stackBufferConveyor2DriveOk AND
    stackBufferConveyor3DriveOk;

stackBufferFull :=
    stackBufferConveyor1StackPresentSensor AND
    stackBufferConveyor2StackPresentSensor AND
    stackBufferConveyor3StackPresentSensor;

rElevatorStackExitClear :=
    elevatorStackExitClearSensor AND elevatorAtMinPosition AND
    NOT elevatorStackExitClearSensorOld;

elevatorStackExitClearSensorOld := elevatorStackExitClearSensor;

tonStackBufferFullSpeedReduction(
    IN := stackBufferFull,
    PT := machineConfig.stackBufferFullSpeedReductionDelay
);

lineSpeedReductionRequest := tonStackBufferFullSpeedReduction.Q;


//==============================================================
// 2) Default outputs
//==============================================================
stackBufferConveyor1Run := FALSE;
stackBufferConveyor2Run := FALSE;
stackBufferConveyor3Run := FALSE;

stackBufferConveyor1SpeedRefMPM := 0.0;
stackBufferConveyor2SpeedRefMPM := 0.0;
stackBufferConveyor3SpeedRefMPM := 0.0;


//==============================================================
// 3) Manual operation
// EN: Manual command ignores the stack presence sensors, but continues
//     to respect the master enable, safety circuit and drive status.
// PT: O comando manual ignora os sensores de presença, mas continua
//     respeitando a habilitação geral, segurança e estado dos drives.
//==============================================================
IF stackBufferConveyorsRunCmd THEN

    stackBufferControlState := 0;
    stackBufferTargetConveyor := 0;

    tonStackBufferStopDelay(IN := FALSE);
    tonStackBufferTransferTimeout(IN := FALSE);

    IF systemRunEnable AND safetyCircuitOk AND allBufferDrivesOk THEN

        stackBufferConveyor1Run := TRUE;
        stackBufferConveyor2Run := TRUE;
        stackBufferConveyor3Run := TRUE;

    END_IF


//==============================================================
// 4) Automatic accumulation
//==============================================================
ELSE

    // EN: A full buffer blocks automatic transfer and stops all conveyors.
    // PT: Buffer cheio bloqueia a transferência automática e para as esteiras.
    IF stackBufferFull OR
       NOT systemRunEnable OR
       NOT safetyCircuitOk OR
       NOT allBufferDrivesOk THEN

        stackBufferControlState := 0;
        stackBufferTargetConveyor := 0;

        tonStackBufferStopDelay(IN := FALSE);
        tonStackBufferTransferTimeout(IN := FALSE);

    ELSE

        CASE stackBufferControlState OF

            0: // IDLE
                tonStackBufferStopDelay(IN := FALSE);
                tonStackBufferTransferTimeout(IN := FALSE);

                IF rElevatorStackExitClear THEN

                    // EN: Always select the furthest available position.
                    // PT: Seleciona sempre a posição livre mais distante.
                    IF NOT stackBufferConveyor3StackPresentSensor THEN
                        stackBufferTargetConveyor := 3;
                        stackBufferControlState := 30;

                    ELSIF NOT stackBufferConveyor2StackPresentSensor THEN
                        stackBufferTargetConveyor := 2;
                        stackBufferControlState := 20;

                    ELSIF NOT stackBufferConveyor1StackPresentSensor THEN
                        stackBufferTargetConveyor := 1;
                        stackBufferControlState := 10;

                    END_IF

                END_IF


            10: // TRANSFER TO BUFFER 1
                stackBufferConveyor1Run := TRUE;

                IF stackBufferConveyor1StackPresentSensor THEN
                    tonStackBufferStopDelay(IN := FALSE);
                    stackBufferControlState := 11;
                END_IF


            11: // BUFFER 1 STOP DELAY
                stackBufferConveyor1Run := TRUE;

                tonStackBufferStopDelay(
                    IN := TRUE,
                    PT := machineConfig.stackBufferConveyorsStopDelay
                );

                IF tonStackBufferStopDelay.Q THEN
                    tonStackBufferStopDelay(IN := FALSE);
                    stackBufferControlState := 0;
                    stackBufferTargetConveyor := 0;
                END_IF


            20: // TRANSFER TO BUFFER 2
                stackBufferConveyor1Run := TRUE;
                stackBufferConveyor2Run := TRUE;

                IF stackBufferConveyor2StackPresentSensor THEN
                    tonStackBufferStopDelay(IN := FALSE);
                    stackBufferControlState := 21;
                END_IF


            21: // BUFFER 2 STOP DELAY
                stackBufferConveyor1Run := TRUE;
                stackBufferConveyor2Run := TRUE;

                tonStackBufferStopDelay(
                    IN := TRUE,
                    PT := machineConfig.stackBufferConveyorsStopDelay
                );

                IF tonStackBufferStopDelay.Q THEN
                    tonStackBufferStopDelay(IN := FALSE);
                    stackBufferControlState := 0;
                    stackBufferTargetConveyor := 0;
                END_IF


            30: // TRANSFER TO BUFFER 3
                stackBufferConveyor1Run := TRUE;
                stackBufferConveyor2Run := TRUE;
                stackBufferConveyor3Run := TRUE;

                // EN: Conveyor 3 stops immediately when its sensor is active.
                // PT: A esteira 3 para imediatamente quando seu sensor é acionado.
                IF stackBufferConveyor3StackPresentSensor THEN
                    stackBufferConveyor1Run := FALSE;
                    stackBufferConveyor2Run := FALSE;
                    stackBufferConveyor3Run := FALSE;

                    stackBufferControlState := 0;
                    stackBufferTargetConveyor := 0;
                END_IF


            ELSE
                stackBufferControlState := 0;
                stackBufferTargetConveyor := 0;

        END_CASE


        //==========================================================
        // 5) Automatic transfer timeout
        //==========================================================
        automaticTransferActive :=
            (stackBufferControlState <> 0);

        tonStackBufferTransferTimeout(
            IN := automaticTransferActive,
            PT := machineConfig.stackBufferTransferTimeout
        );

        IF tonStackBufferTransferTimeout.Q THEN
            stackBufferTransferTimeoutPulse := TRUE;

            tonStackBufferTransferTimeout(IN := FALSE);
            tonStackBufferStopDelay(IN := FALSE);

            stackBufferControlState := 0;
            stackBufferTargetConveyor := 0;

            stackBufferConveyor1Run := FALSE;
            stackBufferConveyor2Run := FALSE;
            stackBufferConveyor3Run := FALSE;
        END_IF

    END_IF

END_IF


//==============================================================
// 6) Sheet stack discharge conveyor coupling
// EN: Run buffer conveyor 1 together with the sheet stack discharge
//     conveyor so the stack is transferred continuously out of the elevator.
//     The existing master, safety and drive interlocks remain active.
// PT: Aciona a esteira buffer 1 junto com a esteira de descarga da pilha
//     para transferir a pilha continuamente para fora do elevador.
//     Os intertravamentos gerais, de segurança e dos drives são mantidos.
//==============================================================
IF sheetStackDischargeConveyorRun AND
   systemRunEnable AND
   safetyCircuitOk AND
   allBufferDrivesOk THEN

    stackBufferConveyor1Run := TRUE;

END_IF;


//==============================================================
// 7) Apply the common fixed speed reference
//==============================================================
IF stackBufferConveyor1Run THEN
    stackBufferConveyor1SpeedRefMPM :=
        machineConfig.stackBufferConveyorsSpeedMPM;
END_IF;

IF stackBufferConveyor2Run THEN
    stackBufferConveyor2SpeedRefMPM :=
        machineConfig.stackBufferConveyorsSpeedMPM;
END_IF;

IF stackBufferConveyor3Run THEN
    stackBufferConveyor3SpeedRefMPM :=
        machineConfig.stackBufferConveyorsSpeedMPM;
END_IF;
END_METHOD

//==============================================================
// COMPLEX STACKER — SYSTEM CONTROL
// EN: Master system run enable and automatic homing requests.
//==============================================================
METHOD _SystemControl

//==============================================================
// 1) Edge detection
//==============================================================
rStartCmd := startCmd AND NOT startCmdOld;
startCmdOld := startCmd;

rStopCmd := stopCmd AND NOT stopCmdOld;
stopCmdOld := stopCmd;



//==============================================================
// 2) Stop machine pulse on critical fault
//==============================================================
// EN: A backstop bypassed in manual remains ignored until the current
//     discharge cycle finishes, even if the selector returns to automatic.
// PT: Um backstop ignorado em manual permanece fora do ciclo até o descarte
//     atual terminar, mesmo que o seletor retorne para automático.
backstopRequiredForAutomaticOperation :=
    backstopAutoCmd AND
    NOT (
        sheetStackDischargeCycleHasManualSkip AND
        (
            sheetStackDischargeActive OR
            sheetStackDischargePending OR
            (sheetStackDischargeControlState <> 0)
        )
    );


stopMachineFaultCondition :=
    NOT safetyCircuitOk OR
    NOT sheetConveyor1DriveOk OR
    NOT sheetConveyor2DriveOk OR
    NOT sheetConveyor3DriveOk OR
    NOT sheetConveyor4DriveOk OR
    (
        backstopRequiredForAutomaticOperation AND
        NOT backstopDriveOk
    ) OR
    NOT elevatorDriveOk OR
    NOT sheetStackDischargeConveyorDriveOk;

rStopMachineFaultCondition :=
    stopMachineFaultCondition AND
    NOT stopMachineFaultConditionOld;

stopMachineFaultConditionOld :=
    stopMachineFaultCondition;

tpStopMachinePulse(
    IN := rStopMachineFaultCondition,
    PT := T#500MS
);

stopMachinePulse :=
    tpStopMachinePulse.Q;


//==============================================================
// 2) Default one-scan requests
//==============================================================
backstopAutoHomeRequest := FALSE;
elevatorAutoHomeRequest := FALSE;


//==============================================================
// 3) Master system run enable
//==============================================================
IF NOT safetyCircuitOk THEN

    systemRunEnable := FALSE;

ELSIF rStopCmd THEN

    systemRunEnable := FALSE;

ELSIF rStartCmd THEN

    systemRunEnable := TRUE;

END_IF;


//==============================================================
// 4) Mandatory reference renewal on every system start
//==============================================================
// EN: A stopped or safety-disabled system cancels pending automatic requests.
//     A new rising edge of startCmd is required before automatic homing.
// PT: O sistema parado ou sem segurança cancela pedidos automáticos pendentes.
//     Uma nova borda de startCmd será necessária antes do homing automático.
IF NOT systemRunEnable THEN

    backstopAutoHomePending := FALSE;
    elevatorAutoHomePending := FALSE;

END_IF;


// EN: Every valid start invalidates the previous position references.
//     An axis already executing homing continues its current cycle.
//     Automatic movement is armed only for axes selected in automatic mode.
// PT: Toda partida válida invalida as referências de posição anteriores.
//     Um eixo que já executa homing continua seu ciclo atual.
//     O movimento automático é armado somente para eixos em modo automático.
IF rStartCmd AND systemRunEnable THEN

    IF NOT (
        (backstopControlState >= 10) AND
        (backstopControlState <= 14)
    ) THEN

        backstopHomed := FALSE;
        backstopInPosition := FALSE;
        backstopAutoHomePending := backstopAutoCmd;

    ELSE

        backstopAutoHomePending := FALSE;

    END_IF;


    IF NOT (
        (elevatorControlState >= 10) AND
        (elevatorControlState <= 14)
    ) THEN

        elevatorHomed := FALSE;
        elevatorReadyForAutomaticCycle := FALSE;
        elevatorInPosition := FALSE;
        elevatorAutoHomePending := elevatorAutoCmd;

    ELSE

        elevatorAutoHomePending := FALSE;

    END_IF;

END_IF;


// EN: Leaving automatic mode cancels automatic movement. The invalidated
//     reference remains invalid until a manual home or a new automatic start.
// PT: Sair do modo automático cancela o movimento automático. A referência
//     invalidada permanece inválida até um home manual ou nova partida automática.
IF NOT backstopAutoCmd THEN
    backstopAutoHomePending := FALSE;
END_IF;

IF NOT elevatorAutoCmd THEN
    elevatorAutoHomePending := FALSE;
END_IF;


//==============================================================
// 5) Release pending homing requests when every permissive is valid
//==============================================================
// EN: The pending memory prevents the start request from being lost while
//     drive-ready, reset or discharge permissives are not yet available.
// PT: A memória pendente evita perder o pedido de partida enquanto os
//     permissivos de drive pronto, reset ou descarte ainda não estão disponíveis.
IF backstopAutoHomePending AND
   systemRunEnable AND
   safetyCircuitOk AND
   backstopAutoCmd AND
   backstopDriveOk AND
   NOT backstopFault AND
   NOT backstopSafeMaxLimit AND
   NOT backstopSafeMinLimit AND
   NOT sheetStackDischargePending AND
   NOT sheetStackDischargeActive AND
   (sheetStackDischargeControlState = 0) THEN

    backstopAutoHomeRequest := TRUE;

END_IF;


IF elevatorAutoHomePending AND
   systemRunEnable AND
   safetyCircuitOk AND
   elevatorAutoCmd AND
   elevatorDriveOk AND
   NOT elevatorFault AND
   NOT elevatorUpperSafetyLimit AND
   NOT elevatorLowerSafetyLimit AND
   NOT sheetStackDischargePending AND
   NOT sheetStackDischargeActive AND
   (sheetStackDischargeControlState = 0) THEN

    elevatorAutoHomeRequest := TRUE;

END_IF;
END_METHOD

END_FUNCTION_BLOCK

// ---- Library/Beckhoff/EL1809/FB_EL1809.TcPOU
FUNCTION_BLOCK FB_EL1809
VAR_INPUT
	


	deviceConfig    : EL1809_DEV_CONFIG; // Configuration settings for the CT121F device
	
	
	
END_VAR
VAR_OUTPUT
		
	digitalInput_01  : BOOL;
	digitalInput_02  : BOOL;
	digitalInput_03  : BOOL;
	digitalInput_04  : BOOL;
	digitalInput_05  : BOOL;
	digitalInput_06  : BOOL;
	digitalInput_07  : BOOL;
	digitalInput_08  : BOOL;
	digitalInput_09  : BOOL;
	digitalInput_10  : BOOL;
	digitalInput_11  : BOOL;
	digitalInput_12  : BOOL;
	digitalInput_13  : BOOL;
	digitalInput_14  : BOOL;
	digitalInput_15  : BOOL;
	digitalInput_16  : BOOL;


END_VAR
VAR
	    PDOS : EL1809_HWTOPLC_PDOS; // Process Data Objects for RWPT01D communication
END_VAR


inputState();

METHOD PRIVATE inputState
// Inputs Mapping Configuration

digitalInput_01 		:= PDOS.digitalInput_00 OR (deviceConfig.enableForce AND deviceConfig.forceDigitalInput_00);
digitalInput_02 		:= PDOS.digitalInput_01 OR (deviceConfig.enableForce AND deviceConfig.forceDigitalInput_01);
digitalInput_03 		:= PDOS.digitalInput_02 OR (deviceConfig.enableForce AND deviceConfig.forceDigitalInput_02);
digitalInput_04 		:= PDOS.digitalInput_03 OR (deviceConfig.enableForce AND deviceConfig.forceDigitalInput_03);
digitalInput_05 		:= PDOS.digitalInput_04 OR (deviceConfig.enableForce AND deviceConfig.forceDigitalInput_04);
digitalInput_06 		:= PDOS.digitalInput_05 OR (deviceConfig.enableForce AND deviceConfig.forceDigitalInput_05);
digitalInput_07	 		:= PDOS.digitalInput_06 OR (deviceConfig.enableForce AND deviceConfig.forceDigitalInput_06);
digitalInput_08 		:= PDOS.digitalInput_07 OR (deviceConfig.enableForce AND deviceConfig.forceDigitalInput_07);
digitalInput_09 		:= PDOS.digitalInput_08 OR (deviceConfig.enableForce AND deviceConfig.forceDigitalInput_08);
digitalInput_10 		:= PDOS.digitalInput_09 OR (deviceConfig.enableForce AND deviceConfig.forceDigitalInput_09);
digitalInput_11 		:= PDOS.digitalInput_10 OR (deviceConfig.enableForce AND deviceConfig.forceDigitalInput_10);
digitalInput_12 		:= PDOS.digitalInput_11 OR (deviceConfig.enableForce AND deviceConfig.forceDigitalInput_11);
digitalInput_13 		:= PDOS.digitalInput_12 OR (deviceConfig.enableForce AND deviceConfig.forceDigitalInput_12);
digitalInput_14 		:= PDOS.digitalInput_13 OR (deviceConfig.enableForce AND deviceConfig.forceDigitalInput_13);
digitalInput_15 		:= PDOS.digitalInput_14 OR (deviceConfig.enableForce AND deviceConfig.forceDigitalInput_14);
digitalInput_16 		:= PDOS.digitalInput_15 OR (deviceConfig.enableForce AND deviceConfig.forceDigitalInput_15);
END_METHOD

END_FUNCTION_BLOCK

// ---- Library/Beckhoff/EL2809/FB_EL2809.TcPOU
FUNCTION_BLOCK FB_EL2809
VAR_INPUT
	


	deviceConfig    : EL2809_DEV_CONFIG; // Configuration settings for the CT222F device
	
	digitalOutput_01 : BOOL;
	digitalOutput_02 : BOOL;
	digitalOutput_03 : BOOL;
	digitalOutput_04 : BOOL;
	digitalOutput_05 : BOOL;
	digitalOutput_06 : BOOL;
	digitalOutput_07 : BOOL;
	digitalOutput_08 : BOOL;
	digitalOutput_09 : BOOL;
	digitalOutput_10 : BOOL;
	digitalOutput_11 : BOOL;
	digitalOutput_12 : BOOL;
	digitalOutput_13 : BOOL;
	digitalOutput_14 : BOOL;
	digitalOutput_15 : BOOL;
	digitalOutput_16 : BOOL;
	
END_VAR
VAR_OUTPUT


END_VAR
VAR
	    PDOS : EL2809_PDOS; // Process Data Objects for RWPT01D communication
END_VAR


outputState();

METHOD PRIVATE outputState
// Outputs Mapping Configuration


PDOS.PlcToHw.digitalOutput_00 := digitalOutput_01 OR (deviceConfig.enableForce AND deviceConfig.forceDigitalOutput_00);
PDOS.PlcToHw.digitalOutput_01 := digitalOutput_02 OR (deviceConfig.enableForce AND deviceConfig.forceDigitalOutput_01);
PDOS.PlcToHw.digitalOutput_02 := digitalOutput_03 OR (deviceConfig.enableForce AND deviceConfig.forceDigitalOutput_02); 
PDOS.PlcToHw.digitalOutput_03 := digitalOutput_04 OR (deviceConfig.enableForce AND deviceConfig.forceDigitalOutput_03); 
PDOS.PlcToHw.digitalOutput_04 := digitalOutput_05 OR (deviceConfig.enableForce AND deviceConfig.forceDigitalOutput_04); 
PDOS.PlcToHw.digitalOutput_05 := digitalOutput_06 OR (deviceConfig.enableForce AND deviceConfig.forceDigitalOutput_05); 
PDOS.PlcToHw.digitalOutput_06 := digitalOutput_07 OR (deviceConfig.enableForce AND deviceConfig.forceDigitalOutput_06); 
PDOS.PlcToHw.digitalOutput_07 := digitalOutput_08 OR (deviceConfig.enableForce AND deviceConfig.forceDigitalOutput_07); 
PDOS.PlcToHw.digitalOutput_08 := digitalOutput_09 OR (deviceConfig.enableForce AND deviceConfig.forceDigitalOutput_08); 
PDOS.PlcToHw.digitalOutput_09 := digitalOutput_10 OR (deviceConfig.enableForce AND deviceConfig.forceDigitalOutput_09); 
PDOS.PlcToHw.digitalOutput_10 := digitalOutput_11 OR (deviceConfig.enableForce AND deviceConfig.forceDigitalOutput_10); 
PDOS.PlcToHw.digitalOutput_11 := digitalOutput_12 OR (deviceConfig.enableForce AND deviceConfig.forceDigitalOutput_11); 
PDOS.PlcToHw.digitalOutput_12 := digitalOutput_13 OR (deviceConfig.enableForce AND deviceConfig.forceDigitalOutput_12); 
PDOS.PlcToHw.digitalOutput_13 := digitalOutput_14 OR (deviceConfig.enableForce AND deviceConfig.forceDigitalOutput_13); 
PDOS.PlcToHw.digitalOutput_14 := digitalOutput_15 OR (deviceConfig.enableForce AND deviceConfig.forceDigitalOutput_14); 
PDOS.PlcToHw.digitalOutput_15 := digitalOutput_16 OR (deviceConfig.enableForce AND deviceConfig.forceDigitalOutput_15);
END_METHOD

END_FUNCTION_BLOCK

// ---- Library/Beckhoff/EL3002 - Ai 2 x 10V - 12bit/FB_EL3002.TcPOU
FUNCTION_BLOCK FB_EL3002
VAR_INPUT PERSISTENT

	deviceConfig    : EL3002_DEV_CONFIG; // Configuration settings for the CT121F device
	
END_VAR
VAR_OUTPUT
		
	Channel1  : REAL;
	Channel2  : REAL;
	
END_VAR
VAR
	    PDOS : EL3002_PDOS; // Process Data Objects for RWPT01D communication
END_VAR


_AnalogInputs();

METHOD PRIVATE _AnalogInputs
VAR_INPUT
END_VAR
// Calculate the actual motor speed
Channel1 := _Scale(
    X := DINT_TO_REAL(PDOS.HwToPLC.Channel1.Value), 
    I_LO := deviceConfig.channel1InputLow, 
    I_HI := deviceConfig.channel1InputHigh, 
    O_LO := deviceConfig.channel1OutputLow, 
    O_HI := deviceConfig.channel1OutputHigh
);

// Calculate the actual motor speed
Channel2 := _Scale(
    X := DINT_TO_REAL(PDOS.HwToPLC.Channel2.Value), 
    I_LO := deviceConfig.channe12InputLow, 
    I_HI := deviceConfig.channe12InputHigh, 
    O_LO := deviceConfig.channe12OutputLow, 
    O_HI := deviceConfig.channe12OutputHigh
);
END_METHOD

METHOD PRIVATE _Scale : REAL
VAR_INPUT
	
	X : REAL;
	I_LO : REAL;
	I_HI : REAL;
	O_LO : REAL;
	O_HI : REAL;
	
END_VAR
IF I_LO = I_HI THEN
	_Scale := O_LO;
ELSE
	_Scale := (O_HI - O_LO) / (I_HI - I_LO) * (LIMIT(I_LO, X, I_HI) - I_LO) + O_LO;
END_IF;
END_METHOD

END_FUNCTION_BLOCK

// ---- Library/Beckhoff/EL4004 - AQ 4 x 0-10V/FB_EL4004.TcPOU
FUNCTION_BLOCK FB_EL4004
VAR_INPUT PERSISTENT

	deviceConfig    : EL4004_DEV_CONFIG; // Configuration settings for the CT121F device
	
END_VAR
VAR_INPUT
		
	Channel1  : REAL;
	Channel2  : REAL;
	Channel3  : REAL;
	Channel4  : REAL;
	
END_VAR
VAR
	    PDOS : EL4004_PDOS; // Process Data Objects for RWPT01D communication
END_VAR

_AnalogOutputs();

METHOD PRIVATE _AnalogOutputs
VAR_INPUT
END_VAR
// Calculate the actual motor speed
PDOS.HwToPLC.Channel1 := REAL_TO_INT(_Scale(
    X	 := Channel1, 
    I_LO := deviceConfig.channel1InputLow, 
    I_HI := deviceConfig.channel1InputHigh, 
    O_LO := deviceConfig.channel1OutputLow, 
    O_HI := deviceConfig.channel1OutputHigh
));
// Calculate the actual motor speed
PDOS.HwToPLC.Channel2 := REAL_TO_INT(_Scale(
    X	 := Channel2, 
    I_LO := deviceConfig.channel2InputLow, 
    I_HI := deviceConfig.channel2InputHigh, 
    O_LO := deviceConfig.channel2OutputLow, 
    O_HI := deviceConfig.channel2OutputHigh
));
// Calculate the actual motor speed
PDOS.HwToPLC.Channel3 := REAL_TO_INT(_Scale(
    X	 := Channel3, 
    I_LO := deviceConfig.channel3InputLow, 
    I_HI := deviceConfig.channel3InputHigh, 
    O_LO := deviceConfig.channel3OutputLow, 
    O_HI := deviceConfig.channel3OutputHigh
));
// Calculate the actual motor speed
PDOS.HwToPLC.Channel4 := REAL_TO_INT(_Scale(
    X	 := Channel4, 
    I_LO := deviceConfig.channel4InputLow, 
    I_HI := deviceConfig.channel4InputHigh, 
    O_LO := deviceConfig.channel4OutputLow, 
    O_HI := deviceConfig.channel4OutputHigh
));
END_METHOD

METHOD PRIVATE _Scale : REAL
VAR_INPUT
	
	X : REAL;
	I_LO : REAL;
	I_HI : REAL;
	O_LO : REAL;
	O_HI : REAL;
	
END_VAR
IF I_LO = I_HI THEN
	_Scale := O_LO;
ELSE
	_Scale := (O_HI - O_LO) / (I_HI - I_LO) * (LIMIT(I_LO, X, I_HI) - I_LO) + O_LO;
END_IF;
END_METHOD

END_FUNCTION_BLOCK

// ---- Library/Beckhoff/EL5152 -2 x  Encoder Input/FB_EL5152.TcPOU
FUNCTION_BLOCK FB_EL5152

//===========================
// INPUTS
//===========================

VAR_INPUT PERSISTENT
	
	channel1DeviceConfig    : EL5152_DEV_CONFIG; // Encoder device configuration (scaling, PPR, timing, etc.)
	channel2DeviceConfig    : EL5152_DEV_CONFIG; // Encoder device configuration (scaling, PPR, timing, etc.)
	
END_VAR

VAR_INPUT
	
	PlcToHw  AT %Q* : EL5152_PLCTOHW; // Output PDOs from PLC to encoder hardware (control signals)
    //==============================================================
    // Channel 1 - set position command
    //==============================================================
    channel1SetPosition     : BOOL;  // Rising edge sets encoder channel 1 position
    channel1DesiredPosition : LREAL; // Desired position in mm for encoder channel 1

    //==============================================================
    // Channel 2 - set position command
    //==============================================================
    channel2SetPosition     : BOOL;  // Rising edge sets encoder channel 2 position
    channel2DesiredPosition : LREAL; // Desired position in mm for encoder channel 2	
	
END_VAR

//===========================
// OUTPUTS
//===========================

VAR_OUTPUT
	
	HwToPlc AT %I* : EL5152_HWTOPLC; // Input PDOs from encoder hardware to PLC (status + values)
	
    channel1EncoderSpeedMMs        : REAL;
    channel1EncoderSpeedMPM        : REAL;
    channel1EncoderSpeedAbsMMs     : REAL;
    channel1EncoderSpeedAbsMPM     : REAL;
    channel1EncoderPosition        : LREAL;
    channel1EncoderModuloPosition  : LREAL;  // Position inside configured modulo range

    channel2EncoderSpeedMMs        : REAL;
    channel2EncoderSpeedMPM        : REAL;
    channel2EncoderSpeedAbsMMs     : REAL;
    channel2EncoderSpeedAbsMPM     : REAL;
    channel2EncoderPosition        : LREAL;
    channel2EncoderModuloPosition  : LREAL;  // Position inside configured modulo range
	
END_VAR
//===========================
// INTERNAL VARIABLES
//===========================

VAR
    //==============================================================
    // Channel 1 - speed calculation memory
    //==============================================================
    instTON_calculateEncSpeedCh1 : TON;

    lastCounterValueCh1          : UDINT;
    counterDeltaCh1              : DINT;
    positionDeltaCh1             : REAL;
    firstCycleCh1                : BOOL := TRUE;

    //==============================================================
    // Channel 2 - speed calculation memory
    //==============================================================
    instTON_calculateEncSpeedCh2 : TON;

    lastCounterValueCh2          : UDINT;
    counterDeltaCh2              : DINT;
    positionDeltaCh2             : REAL;
    firstCycleCh2                : BOOL := TRUE;

    //==============================================================
    // Channel 1 - simulation memory
    //==============================================================
    currentSystemTimeCh1         : ULINT;
    lastCycleTimeCh1             : ULINT;
    deltaTimeMsCh1               : REAL;
    pulsesPerSecondCh1           : REAL;
    pulsesToAddCh1               : DINT;
    simulatedPositionRawValueCh1 : UDINT;
    simulationInitCh1            : BOOL := FALSE;

    //==============================================================
    // Channel 2 - simulation memory
    //==============================================================
    currentSystemTimeCh2         : ULINT;
    lastCycleTimeCh2             : ULINT;
    deltaTimeMsCh2               : REAL;
    pulsesPerSecondCh2           : REAL;
    pulsesToAddCh2               : DINT;
    simulatedPositionRawValueCh2 : UDINT;
    simulationInitCh2            : BOOL := FALSE;

    //==============================================================
    // Set counter command control
    //==============================================================
    setPositionOld               : BOOL;

    instTON_setCounterTimeoutCh1 : TON;
    instTON_setCounterTimeoutCh2 : TON;

    setCounterCommandIssuedCh1   : BOOL := FALSE;
    setCounterCommandIssuedCh2   : BOOL := FALSE;
	
    //==============================================================
    // Channel 1 - set position memory
    //==============================================================
    channel1SetPositionOld       : BOOL;
    channel1SetPositionRawValue  : UDINT;

    //==============================================================
    // Channel 2 - set position memory
    //==============================================================
    channel2SetPositionOld       : BOOL;
    channel2SetPositionRawValue  : UDINT;	
	
END_VAR

//==============================================================
// CHANNEL 1 - Set encoder position
//==============================================================
_SetEncoderPosition(
    channel              := 1,
    setPosition          := channel1SetPosition,
    desiredPosition      := channel1DesiredPosition,
    encoderScalingFactor := channel1DeviceConfig.encoderScalingFactor
);

//==============================================================
// CHANNEL 1 - Modulo position
//==============================================================
channel1EncoderModuloPosition :=
    _CalculateModuloPosition(
        absolutePosition := channel1EncoderPosition,
        moduloPosition   := channel1DeviceConfig.moduloPosition
    );


//==============================================================
// CHANNEL 1 - Position
//==============================================================
channel1EncoderPosition :=
    _CalculateEncoderPositionMM(
        encoderPositionRawValue := HwToPlc.channel1.CounterValue,
        encoderScalingFactor    := channel1DeviceConfig.encoderScalingFactor
    );


//==============================================================
// CHANNEL 1 - Speed
//==============================================================
_CalculateEncoderSpeed(
    channel                   := 1,
    speedCalculationCycleTime := channel1DeviceConfig.speedCalculationCycleTime,
    encoderPositionRawValue   := HwToPlc.channel1.CounterValue,
    encoderScalingFactor      := channel1DeviceConfig.encoderScalingFactor
);


//==============================================================
// CHANNEL 2 - Set encoder position
//==============================================================
_SetEncoderPosition(
    channel              := 2,
    setPosition          := channel2SetPosition,
    desiredPosition      := channel2DesiredPosition,
    encoderScalingFactor := channel2DeviceConfig.encoderScalingFactor
);

//==============================================================
// CHANNEL 2 - Position
//==============================================================
channel2EncoderPosition :=
    _CalculateEncoderPositionMM(
        encoderPositionRawValue := HwToPlc.channel2.CounterValue,
        encoderScalingFactor    := channel2DeviceConfig.encoderScalingFactor
    );
//==============================================================
// CHANNEL 2 - Modulo position
//==============================================================
channel2EncoderModuloPosition :=
    _CalculateModuloPosition(
        absolutePosition := channel2EncoderPosition,
        moduloPosition   := channel2DeviceConfig.moduloPosition
    );

//==============================================================
// CHANNEL 2 - Speed
//==============================================================
_CalculateEncoderSpeed(
    channel                   := 2,
    speedCalculationCycleTime := channel2DeviceConfig.speedCalculationCycleTime,
    encoderPositionRawValue   := HwToPlc.channel2.CounterValue,
    encoderScalingFactor      := channel2DeviceConfig.encoderScalingFactor
);

METHOD PRIVATE _CalculateEncoderPositionMM : LREAL
// ==============================================================================
// Calculates the absolute encoder position in millimeters
// using the raw counter value and a scaling factor.
// ==============================================================================

VAR_INPUT
    encoderPositionRawValue : UDINT; // Raw counter value from encoder
    encoderScalingFactor    : REAL;  // Scale factor: mm per pulse
END_VAR
// Convert raw encoder counter value to engineering position using scaling factor
_CalculateEncoderPositionMM := UDINT_TO_LREAL(encoderPositionRawValue) * REAL_TO_LREAL(encoderScalingFactor);
END_METHOD

METHOD PRIVATE _CalculateEncoderSpeed
// ==================================================================================================
// Calculates encoder speed in both mm/s and m/min for channel 1 or channel 2.
//
// IMPORTANT:
// Each channel has independent timer, previous counter value and first-cycle flag.
// ==================================================================================================

VAR_INPUT
    channel                   : USINT; // 1 = Channel 1, 2 = Channel 2
    speedCalculationCycleTime : TIME;  // Time interval for speed calculation
    encoderPositionRawValue   : UDINT; // Current raw value from encoder counter
    encoderScalingFactor      : REAL;  // Scaling factor: mm per encoder pulse
END_VAR

VAR
    calculationTimeSec : REAL;
END_VAR


// Convert configured calculation time from milliseconds to seconds
calculationTimeSec := TIME_TO_REAL(speedCalculationCycleTime) / 1000.0;

IF calculationTimeSec <= 0.0 THEN
    RETURN;
END_IF


CASE channel OF

    //==============================================================
    // CHANNEL 1
    //==============================================================
    1:
        instTON_calculateEncSpeedCh1(IN := TRUE, PT := speedCalculationCycleTime);

        IF instTON_calculateEncSpeedCh1.Q THEN
            // Reset timer
            instTON_calculateEncSpeedCh1(IN := FALSE);

            IF NOT firstCycleCh1 THEN

